// TwinCAT 3 PLC project TcUnit_Learning_Space
// ProgramVersion: 3.1.4024.0
// libraries:
//   Tc2_Standard, * (Beckhoff Automation GmbH)
//   Tc2_System, * (Beckhoff Automation GmbH)
//   Tc3_Module, * (Beckhoff Automation GmbH)
//   TcUnit, * (www.tcunit.org)
// project tree:
//   Classes/ MyCalculatorClass.TcPOU
//   / PlcTask.TcTTO
//   POUs/ MAIN.TcPOU
//   TestSuites/ MyCalculatorTests.TcPOU
// real-time tasks:
//   TASK PlcTask: cycle T#10ms, priority 20, ADS port 350
//   TASK PlcTask1: cycle T#10ms, priority 21, ADS port 351
//   TASK PlcTask2: cycle T#10ms, priority 22, ADS port 352

CONFIGURATION TcUnit_Learning_Space
    RESOURCE PLC ON TwinCAT3
        TASK PlcTask(INTERVAL := T#10ms, PRIORITY := 20);
        PROGRAM MAIN WITH PlcTask : MAIN;
    END_RESOURCE
END_CONFIGURATION

// ---- POUs/MAIN.TcPOU
PROGRAM MAIN
VAR
	fbCalcTest : MyCalculatorTests;
END_VAR

TcUnit.RUN();

END_PROGRAM

// ---- TestSuites/MyCalculatorTests.TcPOU
FUNCTION_BLOCK MyCalculatorTests EXTENDS FB_TestSuite
VAR_INPUT
END_VAR
VAR_OUTPUT
END_VAR
VAR
END_VAR

DivideByZeroTest();
TwoPositiveIntegers();

METHOD DivideByZeroTest : REFERENCE TO FB_Test
VAR
	myCalc : MyCalculatorClass;
    Result : UINT;
    ExpectedSum : UINT := 4;
END_VAR
TEST('GivenAZeroDivisorThenTheCalcShouldReturnAError');
 
Result :=  myCalc.Divide(2,0);

AssertEquals(Expected := ExpectedSum,
             Actual := Result,
             Message := 'The division didnt return an error');
 
TEST_FINISHED();
END_METHOD

METHOD TwoPositiveIntegers : REFERENCE TO FB_Test
VAR
	myCalc : MyCalculatorClass;
    Result : INT;
    ExpectedSum : INT := 2;
END_VAR
TEST('GivenTwoPositiveIntegersThenTheResultShouldBeValid');
 
Result := myCalc.Divide(4,2);
 
AssertEquals(Expected := ExpectedSum,
             Actual := Result,
             Message := 'The division returned an error');
 
TEST_FINISHED();
END_METHOD

END_FUNCTION_BLOCK

// ---- Classes/MyCalculatorClass.TcPOU
FUNCTION_BLOCK MyCalculatorClass
VAR
END_VAR

METHOD Divide : INT
VAR_INPUT
	x : INT;
	y : INT;
END_VAR
IF y <> 0 THEN
	Divide := x/y;
ELSE
	Divide := -1;
END_IF
END_METHOD

END_FUNCTION_BLOCK
